{attribute 'qualified_only'}
VAR_GLOBAL
	bRunStopToSafety 	AT %Q*	: BOOL := TRUE;
	bErrAck			 	AT %Q*	: BOOL;
END_VAR

(* stored: Version 1.1.0.1
   GVL GVL_Safety: Id {0e0c9c48-4076-4609-b771-0ecf29577e5d} *)
